// TIA Portal V20 export
DATA_BLOCK "InstInterfaceSignals"   // DB39
{ DB_Accessible_From_OPC_UA := 'FALSE' }
AUTHOR : SICAR
FAMILY : Diag
VERSION : 1.0
// stored: DBAccessibleFromOPCUA false, DBAccessibleFromWebserver false, InstanceOfName CallInterfaceSignals, InstanceOfType FB
"CallInterfaceSignals"
   // VAR
   //    statReadValueHmi : Bool;
   //    statSelectSignalsHmi : USInt;
   //    statSelectSignalsOld { ExternalAccessible := 'False'; ExternalVisible := 'False'; ExternalWritable := 'False'} : USInt;
   //    statRisEdgeReadName { ExternalAccessible := 'False'; ExternalVisible := 'False'; ExternalWritable := 'False'} : Bool;
   //    statPosPulseReadName : Bool;
   // END_VAR
   // VAR RETAIN
   //    statInterfaceSignalsHmi : Array[0..70] of "typeInterfaceSignalsHmi";
   // END_VAR
   // VAR
   //    instSignalsLeft { ExternalAccessible := 'False'; ExternalVisible := 'False'; ExternalWritable := 'False'} : Array[0..70] of "LAF_InterfaceSignalsBool";
   //    instSignalsRight { ExternalAccessible := 'False'; ExternalVisible := 'False'; ExternalWritable := 'False'} : Array[0..70] of "LAF_InterfaceSignalsBool";
   // END_VAR
BEGIN
   statInterfaceSignalsHmi[1].valueSymbolLeft.freeDescriptionText := WSTRING#'ReelCut To STK30';
   statInterfaceSignalsHmi[2].valueSymbolLeft.freeDescriptionText := WSTRING#'ReelCut to STK40';
   statInterfaceSignalsHmi[3].valueSymbolLeft.freeDescriptionText := WSTRING#'BK01';
   statInterfaceSignalsHmi[4].valueSymbolLeft.freeDescriptionText := WSTRING#'BK02';
   statInterfaceSignalsHmi[5].valueSymbolLeft.freeDescriptionText := WSTRING#'BK03';
   statInterfaceSignalsHmi[6].valueSymbolLeft.freeDescriptionText := WSTRING#'BK04';
   statInterfaceSignalsHmi[7].valueSymbolLeft.freeDescriptionText := WSTRING#'BK05';
   statInterfaceSignalsHmi[8].valueSymbolLeft.freeDescriptionText := WSTRING#'BK06';
   statInterfaceSignalsHmi[9].valueSymbolLeft.freeDescriptionText := WSTRING#'BK07';
   statInterfaceSignalsHmi[10].valueSymbolLeft.freeDescriptionText := WSTRING#'BK08';
   statInterfaceSignalsHmi[11].valueSymbolLeft.freeDescriptionText := WSTRING#'BK09';
   statInterfaceSignalsHmi[12].valueSymbolLeft.freeDescriptionText := WSTRING#'BK10';
   statInterfaceSignalsHmi[13].valueSymbolLeft.freeDescriptionText := WSTRING#'SBK01';
   statInterfaceSignalsHmi[14].valueSymbolLeft.freeDescriptionText := WSTRING#'SBK02';
   statInterfaceSignalsHmi[15].valueSymbolLeft.freeDescriptionText := WSTRING#'SBK03';
   statInterfaceSignalsHmi[16].valueSymbolLeft.freeDescriptionText := WSTRING#'SBK04';
   statInterfaceSignalsHmi[17].valueSymbolLeft.freeDescriptionText := WSTRING#'SBK05';
   statInterfaceSignalsHmi[18].valueSymbolLeft.freeDescriptionText := WSTRING#'SBK06';
   statInterfaceSignalsHmi[19].valueSymbolLeft.freeDescriptionText := WSTRING#'SBK01';
   statInterfaceSignalsHmi[20].valueSymbolLeft.freeDescriptionText := WSTRING#'SBK02';
   statInterfaceSignalsHmi[21].valueSymbolLeft.freeDescriptionText := WSTRING#'SBK03';
   statInterfaceSignalsHmi[22].valueSymbolLeft.freeDescriptionText := WSTRING#'SBK04';
   statInterfaceSignalsHmi[23].valueSymbolLeft.freeDescriptionText := WSTRING#'SBK05';
   statInterfaceSignalsHmi[24].valueSymbolLeft.freeDescriptionText := WSTRING#'SBK06';
   statInterfaceSignalsHmi[25].valueSymbolLeft.freeDescriptionText := WSTRING#'SBK07';
   statInterfaceSignalsHmi[26].valueSymbolLeft.freeDescriptionText := WSTRING#'SBK08';
   statInterfaceSignalsHmi[27].valueSymbolLeft.freeDescriptionText := WSTRING#'SBK09';
   statInterfaceSignalsHmi[28].valueSymbolLeft.freeDescriptionText := WSTRING#'PM01';
   statInterfaceSignalsHmi[29].valueSymbolLeft.freeDescriptionText := WSTRING#'PM02';
   statInterfaceSignalsHmi[30].valueSymbolLeft.freeDescriptionText := WSTRING#'PM03';
   statInterfaceSignalsHmi[31].valueSymbolLeft.freeDescriptionText := WSTRING#'PM04';
   statInterfaceSignalsHmi[37].valueSymbolLeft.freeDescriptionText := WSTRING#'SP501';
   statInterfaceSignalsHmi[38].valueSymbolLeft.freeDescriptionText := WSTRING#'SP502';
   statInterfaceSignalsHmi[39].valueSymbolLeft.freeDescriptionText := WSTRING#'SP503';
   statInterfaceSignalsHmi[40].valueSymbolLeft.freeDescriptionText := WSTRING#'SP504';
   statInterfaceSignalsHmi[41].valueSymbolLeft.freeDescriptionText := WSTRING#'SP505';
   statInterfaceSignalsHmi[42].valueSymbolLeft.freeDescriptionText := WSTRING#'SP506';
   statInterfaceSignalsHmi[43].valueSymbolLeft.freeDescriptionText := WSTRING#'SP507';
   statInterfaceSignalsHmi[44].valueSymbolLeft.freeDescriptionText := WSTRING#'SP508';
   statInterfaceSignalsHmi[45].valueSymbolLeft.freeDescriptionText := WSTRING#'SP509';
   statInterfaceSignalsHmi[46].valueSymbolLeft.freeDescriptionText := WSTRING#'SP510';
   statInterfaceSignalsHmi[47].valueSymbolLeft.freeDescriptionText := WSTRING#'SP511';
   statInterfaceSignalsHmi[48].valueSymbolLeft.freeDescriptionText := WSTRING#'SP512';
   statInterfaceSignalsHmi[1].valueSymbolRight.freeDescriptionText := WSTRING#'ReelCut To STK30';
   statInterfaceSignalsHmi[2].valueSymbolRight.freeDescriptionText := WSTRING#'ReelCut to STK40';
   statInterfaceSignalsHmi[3].valueSymbolRight.freeDescriptionText := WSTRING#'BK01';
   statInterfaceSignalsHmi[4].valueSymbolRight.freeDescriptionText := WSTRING#'BK02';
   statInterfaceSignalsHmi[5].valueSymbolRight.freeDescriptionText := WSTRING#'BK03';
   statInterfaceSignalsHmi[6].valueSymbolRight.freeDescriptionText := WSTRING#'BK04';
   statInterfaceSignalsHmi[7].valueSymbolRight.freeDescriptionText := WSTRING#'BK05';
   statInterfaceSignalsHmi[8].valueSymbolRight.freeDescriptionText := WSTRING#'BK06';
   statInterfaceSignalsHmi[9].valueSymbolRight.freeDescriptionText := WSTRING#'BK07';
   statInterfaceSignalsHmi[10].valueSymbolRight.freeDescriptionText := WSTRING#'BK08';
   statInterfaceSignalsHmi[11].valueSymbolRight.freeDescriptionText := WSTRING#'BK09';
   statInterfaceSignalsHmi[12].valueSymbolRight.freeDescriptionText := WSTRING#'BK10';
   statInterfaceSignalsHmi[13].valueSymbolRight.freeDescriptionText := WSTRING#'SBK01';
   statInterfaceSignalsHmi[14].valueSymbolRight.freeDescriptionText := WSTRING#'SBK02';
   statInterfaceSignalsHmi[15].valueSymbolRight.freeDescriptionText := WSTRING#'SBK03';
   statInterfaceSignalsHmi[16].valueSymbolRight.freeDescriptionText := WSTRING#'SBK04';
   statInterfaceSignalsHmi[17].valueSymbolRight.freeDescriptionText := WSTRING#'SBK05';
   statInterfaceSignalsHmi[18].valueSymbolRight.freeDescriptionText := WSTRING#'SBK06';
   statInterfaceSignalsHmi[19].valueSymbolRight.freeDescriptionText := WSTRING#'SBK01';
   statInterfaceSignalsHmi[20].valueSymbolRight.freeDescriptionText := WSTRING#'SBK02';
   statInterfaceSignalsHmi[21].valueSymbolRight.freeDescriptionText := WSTRING#'SBK03';
   statInterfaceSignalsHmi[22].valueSymbolRight.freeDescriptionText := WSTRING#'SBK04';
   statInterfaceSignalsHmi[23].valueSymbolRight.freeDescriptionText := WSTRING#'SBK05';
   statInterfaceSignalsHmi[24].valueSymbolRight.freeDescriptionText := WSTRING#'SBK06';
   statInterfaceSignalsHmi[25].valueSymbolRight.freeDescriptionText := WSTRING#'SBK07';
   statInterfaceSignalsHmi[26].valueSymbolRight.freeDescriptionText := WSTRING#'SBK08';
   statInterfaceSignalsHmi[27].valueSymbolRight.freeDescriptionText := WSTRING#'SBK09';
   statInterfaceSignalsHmi[28].valueSymbolRight.freeDescriptionText := WSTRING#'PM01';
   statInterfaceSignalsHmi[29].valueSymbolRight.freeDescriptionText := WSTRING#'PM02';
   statInterfaceSignalsHmi[30].valueSymbolRight.freeDescriptionText := WSTRING#'PM03';
   statInterfaceSignalsHmi[31].valueSymbolRight.freeDescriptionText := WSTRING#'PM04';
   statInterfaceSignalsHmi[37].valueSymbolRight.freeDescriptionText := WSTRING#'SP501';
   statInterfaceSignalsHmi[38].valueSymbolRight.freeDescriptionText := WSTRING#'SP502';
   statInterfaceSignalsHmi[39].valueSymbolRight.freeDescriptionText := WSTRING#'SP503';
   statInterfaceSignalsHmi[40].valueSymbolRight.freeDescriptionText := WSTRING#'SP504';
   statInterfaceSignalsHmi[41].valueSymbolRight.freeDescriptionText := WSTRING#'SP505';
   statInterfaceSignalsHmi[42].valueSymbolRight.freeDescriptionText := WSTRING#'SP506';
   statInterfaceSignalsHmi[43].valueSymbolRight.freeDescriptionText := WSTRING#'SP507';
   statInterfaceSignalsHmi[44].valueSymbolRight.freeDescriptionText := WSTRING#'SP508';
   statInterfaceSignalsHmi[45].valueSymbolRight.freeDescriptionText := WSTRING#'SP509';
   statInterfaceSignalsHmi[46].valueSymbolRight.freeDescriptionText := WSTRING#'SP510';
   statInterfaceSignalsHmi[47].valueSymbolRight.freeDescriptionText := WSTRING#'SP511';
   statInterfaceSignalsHmi[48].valueSymbolRight.freeDescriptionText := WSTRING#'SP512';
END_DATA_BLOCK
